// TwinCAT 3 PLC project PLC
// ProgramVersion: 3.1.4024.0
// libraries:
//   EfficientIO Communicator, * (EfficientIO)
//   Lynus Energy Basic, * (Lynus AG)
//   Tc2_Standard, * (Beckhoff Automation GmbH)
//   Tc2_System, * (Beckhoff Automation GmbH)
//   Tc3_Module, * (Beckhoff Automation GmbH)
// project tree:
//   / FastTask.TcTTO, MiddleTask.TcTTO, SlowTask.TcTTO
//   POUs/ prgCom.TcPOU (not stored), prgMain.TcPOU, prgRWEffIO.TcPOU (not stored), prgVarEffIO.TcPOU
// real-time tasks:
//   TASK PlcTask: cycle T#10ms, priority 20, ADS port 350
//   TASK FastTask: cycle T#10ms, priority 21, ADS port 351
//   TASK MiddleTask: cycle T#10ms, priority 22, ADS port 352
//   TASK SlowTask: cycle T#10ms, priority 23, ADS port 353
// I/O:
//   DEVICE Gerät 2 (CX-BK)
//     Box 1 (CX-BK)
// variable links:
//   PLC/PLC Instance <-> Device 2 (CX-BK)/Box 1 (CX-BK)
//     MiddleTask Inputs/prgMain.m_In1 <-> Term 3 (KL1408)/Channel 1/Eingang
//     MiddleTask Inputs/prgMain.m_In2 <-> Term 3 (KL1408)/Channel 2/Eingang
//     MiddleTask Outputs/prgMain.m_out1 <-> Term 2 (KL2408)/Channel 1/Ausgang

CONFIGURATION PLC
    RESOURCE PLC ON TwinCAT3
        TASK FastTask(INTERVAL := T#10ms, PRIORITY := 21);
        TASK MiddleTask(INTERVAL := T#10ms, PRIORITY := 22);
        TASK SlowTask(INTERVAL := T#10ms, PRIORITY := 23);
        PROGRAM prgRWEffIO WITH FastTask : prgRWEffIO;
        PROGRAM prgVarEffIO WITH FastTask : prgVarEffIO;
        PROGRAM prgMain WITH MiddleTask : prgMain;
        PROGRAM prgCom WITH SlowTask : prgCom;
    END_RESOURCE
END_CONFIGURATION

// ---- POUs/prgVarEffIO.TcPOU
PROGRAM prgVarEffIO
VAR
	fbVar		: FB_VarInfo_V3;
END_VAR

fbVar(
	bReadInfo:= , 
	eTMCFile:= eSelectTMCFile.eDontUseTMCFile, 
	eSavePositionTMCFile:= eSavePositionOnPLC.ePostionHardDisk, 
	udiCounterFoundVariables=> , 
	bError=> , 
	bBusy=> , 
	byProgress=> , 
	udiErrorCodeOut=> , 
	eErrorVarInfo_Out=> , 
	sVarWithError=> );
fbVar(
	bReadInfo:= , 
	eTMCFile:= eSelectTMCFile.eDontUseTMCFile, 
	eSavePositionTMCFile:= eSavePositionOnPLC.ePostionHardDisk, 
	udiCounterFoundVariables=> , 
	bError=> , 
	bBusy=> , 
	byProgress=> , 
	udiErrorCodeOut=> , 
	eErrorVarInfo_Out=> , 
	sVarWithError=> );
fbVar(
	bReadInfo:= , 
	eTMCFile:= eSelectTMCFile.eDontUseTMCFile, 
	eSavePositionTMCFile:= eSavePositionOnPLC.ePostionHardDisk, 
	udiCounterFoundVariables=> , 
	bError=> , 
	bBusy=> , 
	byProgress=> , 
	udiErrorCodeOut=> , 
	eErrorVarInfo_Out=> , 
	sVarWithError=> );

END_PROGRAM

// ---- POUs/prgMain.TcPOU
PROGRAM prgMain
VAR
	m_Command_Knetzgau_RESET					: BOOL;							//{#lynus.ag#()}
	m_out1								AT%Q* 	: BOOL;
	m_In1								AT%I* 	: BOOL;
	m_In2								AT%I* 	: BOOL;
	m_Input_Beacon_Knetzgau						: BOOL;							//{#lynus.ag#()}
	m_Input_Siren_Knetzgau						: BOOL;							//{#lynus.ag#()}
	r_tigt_Start_Reset: R_trig;
	tof_Reset: Tof;
	m_LiveBit_5min_Knetzgau						: BOOL;							//{#lynus.ag#()}
	ton_5Min: Ton;
END_VAR

r_tigt_Start_Reset( CLK := m_Command_Knetzgau_RESET);

tof_Reset(	IN:= r_tigt_Start_Reset.Q, 
			PT:= T#2S , 
			Q=> m_out1, 
			ET=> );

 m_Input_Beacon_Knetzgau		:= 			m_In1;
 m_Input_Siren_Knetzgau			:= 			m_In2;		// nicht ausgeführt
 
  ton_5Min(	In := NOT ton_5min.Q	,
	 		PT := T#5M);
			
IF ton_5min.Q AND m_LiveBit_5min_Knetzgau THEN
	m_LiveBit_5min_Knetzgau := FALSE;
ELSIF  ton_5min.Q AND NOT m_LiveBit_5min_Knetzgau THEN
	m_LiveBit_5min_Knetzgau := TRUE;
END_IF

END_PROGRAM
